PROGRAM P42_BrakeControl
VAR
	fbTOF_MotorBrake: TOF;
	OnHome : BOOL;
	HomeSwitchPositionON : DINT;
	enablecounter : DINT;
	HomeSwitchPositionOff : DINT;
	
	
END_VAR

(*
//*****************************************************************Notes**********************************************************\\


  
  
//*****************************************************************Revs**********************************************************\\
   (          who            )(    Date    ) (   Rev     ) (								Disc						)
     Chris Mauban			 	2016.05.05		0.00.01		Added Brake Logic for Load Brake
	 Brent Miller				2016.05.25		  0.00.02		Changed Motor Brake Logic to include a wait command before disabling motor			
     		 								 				
	 						
	
//*****************************************************************Code**********************************************************\\
*)



//Brake Logic for Motor brake	

// To DO:  	For Motor brake logic, brake should release once the drive has enabled and is energized
//			Brake should engage when Deadman button is released, wait 0.5 sec then disable the motor

		
		IF  GVL_Modes.bDrive_Enable AND kidaxis.Status.STATso AND kidaxis.status.ready THEN
				GVL_DriveParameters.controlWord := 15;
				GVL_Safe_IO.bRelease_Load_Brake := TRUE;
				IF  GVL_Hardware_IO.bLoad_Brake_Feedback THEN
					EnableCounter := ENableCounter + 1;
				END_IF
				IF EnableCounter > 50 THEN 
					GVL_Safe_IO.bRelease_Motor_Brake := TRUE;
			 		EnableCounter := 50; 
				END_IF
		ELSE
				IF EnableCounter > 0 THEN enablecounter :=0; END_IF
				GVL_Safe_IO.bRelease_Motor_Brake := FALSE;
				enablecounter := enablecounter -1;
				IF enablecounter < -50 THEN  
					enablecounter := -50; 
					IF  kidaxis.Status.STATso THEN GVL_DriveParameters.controlWord := 7; END_IF
				END_IF
		END_IF
		

IF NOT GVL_Safe_IO.bContactor  THEN GVL_Safe_IO.bRelease_Load_Brake := FALSE; GVL_Safe_IO.bRelease_Motor_Brake := FALSE; END_IF


//Brake Logic for Load Brake
//IF NOT GVL_PLC.bGlobal_Error THEN
//	GVL_Safe_IO.bRelease_Load_Brake := TRUE;
//ELSE
//	GVL_Safe_IO.bRelease_Load_Brake := FALSE;
//END_IF

IF GVL_Safe_IO.bCross_Groove AND NOT OnHome THEN
	HomeSwitchPositionON := KidAxis.actualPos;
	OnHome := TRUE;
ELSIF NOT GVL_SAFE_IO.bCross_Groove AND ONHOME THEN
	HomeSwitchPositionOFF := KidAxis.actualPos;
	OnHome := FALSE;
END_IF
kidAxis.CheckIn.Home_Tripped := OnHome;

ACTION A1_BrakeTest:
(*
	This program will allow the technician to test the functionality of each of the brakes.
	When in "Test" mode, both brakes will engage (not-energized) regardless of system status
	- operator will then be allowed to manually release one brake at a time (momentary release). This allows the operator to check functionality & load holding ability
	- 

*)
END_ACTION

END_PROGRAM

(* stored: Version 1.1.0.1, ProductVersion 3.1.4022.7
   POU P42_BrakeControl: Id {a10ecb5a-62f5-43ed-818f-4cf8d35aaccc}, SpecialFunc None
   Action A1_BrakeTest: Id {294c3341-0a5c-4117-bed7-3ab823497808} *)
